(* IEC 61131-3 sources: eCockpitGit/test_project/src/%F%00 Library/%F%Common Functions/%F%Dynamic Array/%F%Dynamic Array Helpers, 6 files *)

(* ---- %POU%FU_dynamicModuleArrayFromStruct.st ---- *)
FUNCTION FU_dynamicModuleArrayFromStruct : SLMResult
VAR_INPUT
	dynArrHandler		:REFERENCE TO FB_DynamicArray;
	reader				:ITF_StructReaderBase;
END_VAR
VAR
	length				:WORD;
	i					:WORD;
	buffer				:POINTER TO FB_Module;
END_VAR
(*%!%__DELIMITER__%!%*)
IF reader.valueType = EStructType.tArray THEN
	dynArrHandler.empty();
	reader.enterObjectArray();
	length											:=		reader.amountInSelection;
	FU_dynamicModuleArrayFromStruct					:=		dynArrHandler.allocate(size:=length);
	IF FU_dynamicModuleArrayFromStruct.success AND length > 0 THEN
		FOR i := 1 TO length DO
			IF reader.nextArray() <> EStructType.none THEN
				buffer								:=		GMod.modMan.getModuleByUID(modUID:=reader.readWord());
				IF buffer <> 0 THEN
					FU_dynamicModuleArrayFromStruct	:=		dynArrHandler.appendElement(element:=ADR(buffer),elementSize:=SIZEOF(buffer));
					IF NOT(FU_dynamicModuleArrayFromStruct.success) THEN
						EXIT;
					END_IF
				END_IF
			ELSE
				EXIT;
			END_IF
		END_FOR
	END_IF
	reader.exitObjectArray();
END_IF

(* ---- %POU%FU_dynamicModuleArrayToStruct.st ---- *)
FUNCTION FU_dynamicModuleArrayToStruct : SLMResult
VAR_INPUT
	dynArrHandler		:REFERENCE TO FB_DynamicArray;
	writer				:ITF_StructWriterBase;
END_VAR
VAR
	i					:WORD;
	buffer				:POINTER TO FB_Module;
END_VAR
(*%!%__DELIMITER__%!%*)
writer.arrayStart(singleLine:=TRUE);
IF dynArrHandler.S_lenght > 0 THEN
	FOR i := 0 TO dynArrHandler.S_lenght - 1 DO
		dynArrHandler.getElementByIndex(element:=ADR(buffer),elementSize:=SIZEOF(buffer),index:=i);
		writer.writeDint(value:=buffer^._UID);
	END_FOR
END_IF
writer.structEnd();

(* ---- %POU%FU_dynamicUIDArrayFromStruct.st ---- *)
FUNCTION FU_dynamicUIDArrayFromStruct : SLMResult
VAR_INPUT
	dynArrHandler		:REFERENCE TO FB_DynamicArray;
	reader				:ITF_StructReaderBase;
END_VAR
VAR
	length				:WORD;
	i					:WORD;
	buffer				:AModuleUID;
END_VAR
(*%!%__DELIMITER__%!%*)
IF reader.valueType = EStructType.tArray THEN
	dynArrHandler.empty();
	reader.enterObjectArray();
	length											:=		reader.amountInSelection;
	FU_dynamicUIDArrayFromStruct					:=		dynArrHandler.allocate(size:=length);
	IF FU_dynamicUIDArrayFromStruct.success AND length > 0 THEN
		FOR i := 1 TO length DO
			IF reader.nextArray() <> EStructType.none THEN
				buffer								:=		reader.readWord();
				FU_dynamicUIDArrayFromStruct		:=		dynArrHandler.appendElement(element:=ADR(buffer),elementSize:=SIZEOF(buffer));
				IF NOT(FU_dynamicUIDArrayFromStruct.success) THEN
					EXIT;
				END_IF
			ELSE
				EXIT;
			END_IF
		END_FOR
	END_IF
	reader.exitObjectArray();
END_IF

(* ---- %POU%FU_dynamicUIDArrayToStruct.st ---- *)
FUNCTION FU_dynamicUIDArrayToStruct : SLMResult
VAR_INPUT
	dynArrHandler		:REFERENCE TO FB_DynamicArray;
	writer				:ITF_StructWriterBase;
END_VAR
VAR
	i					:WORD;
	buffer				:AModuleUID;
END_VAR
(*%!%__DELIMITER__%!%*)
writer.arrayStart(singleLine:=TRUE);
IF dynArrHandler.S_lenght > 0 THEN
	FOR i := 0 TO dynArrHandler.S_lenght - 1 DO
		dynArrHandler.getElementByIndex(element:=ADR(buffer),elementSize:=SIZEOF(buffer),index:=i);
		writer.writeDint(value:=buffer);
	END_FOR
END_IF
writer.structEnd();

(* ---- %POU%FU_dynamicWordArrayFromStruct.st ---- *)
FUNCTION FU_dynamicWordArrayFromStruct : SLMResult
VAR_INPUT
	dynArrHandler		:REFERENCE TO FB_DynamicArray;
	reader				:ITF_StructReaderBase;
END_VAR
VAR
	length				:WORD;
	i					:WORD;
	buffer				:WORD;
END_VAR
(*%!%__DELIMITER__%!%*)
IF reader.valueType = EStructType.tArray THEN
	dynArrHandler.empty();
	reader.enterObjectArray();
	length										:=		reader.amountInSelection;
	FU_dynamicWordArrayFromStruct				:=		dynArrHandler.allocate(size:=length);
	IF FU_dynamicWordArrayFromStruct.success AND length > 0 THEN
		FOR i := 1 TO length DO
			IF reader.nextArray() <> EStructType.none THEN
				buffer							:=		reader.readWord();
				FU_dynamicWordArrayFromStruct	:=		dynArrHandler.appendElement(element:=ADR(buffer),elementSize:=SIZEOF(buffer));
				IF NOT(FU_dynamicWordArrayFromStruct.success) THEN
					EXIT;
				END_IF
			ELSE
				EXIT;
			END_IF
		END_FOR
	END_IF
	reader.exitObjectArray();
END_IF

(* ---- %POU%FU_dynamicWordArrayToStruct.st ---- *)
FUNCTION FU_dynamicWordArrayToStruct : SLMResult
VAR_INPUT
	dynArrHandler		:REFERENCE TO FB_DynamicArray;
	writer				:ITF_StructWriterBase;
END_VAR
VAR
	i					:WORD;
	buffer				:WORD;
END_VAR
(*%!%__DELIMITER__%!%*)
writer.arrayStart(singleLine:=TRUE);
IF dynArrHandler.S_lenght > 0 THEN
	FOR i := 0 TO dynArrHandler.S_lenght - 1 DO
		dynArrHandler.getElementByIndex(element:=ADR(buffer),elementSize:=SIZEOF(buffer),index:=i);
		writer.writeDint(value:=buffer);
	END_FOR
END_IF
writer.structEnd();
